// TIA Portal V20 export
VAR_GLOBAL   // PLC tag table "LConSMC_Configuration"
END_VAR
VAR_GLOBAL CONSTANT   // user constants
   LCON_VELO_MONITORING_ADJUSTMENT_PERCENT : LReal := 20.0;   // [%] Maximum velocity deviation to detect drive runaway in torque controlled modes. Value is a percentage value of the active velocity override
END_VAR
